(* -----------------------------------------------------------------------------
| This sample has been supplied by Beckhoff As-Is and is intended only as an   |
| example implementation. Functionality is not guaranteed.                     |
----------------------------------------------------------------------------- *)

FUNCTION_BLOCK FB_CorkingRotation
VAR_INPUT
	bExecute : BOOL;
	bLimitSwitch : BOOL;
END_VAR
VAR_OUTPUT
	bRotation : BOOL; 
	bDone : BOOL;
	bError : BOOL;
	nErrId : UDINT;
END_VAR
VAR
	nCnt : UDINT;
END_VAR

(* -----------------------------------------------------------------------------
| This sample has been supplied by Beckhoff As-Is and is intended only as an   |
| example implementation. Functionality is not guaranteed.                     |
----------------------------------------------------------------------------- *)

IF bExecute THEN
	nCnt := nCnt + 1;
	bRotation := (nCnt >= 1 AND nCnt < 100) OR
				(nCnt >= 201 AND nCnt < 300) OR
				(nCnt >= 401 AND nCnt < 500) OR
				(nCnt >= 601 AND nCnt < 700) OR
				(nCnt >= 800 AND nCnt < 1000);
	IF nCnt >= 1000 THEN
		IF bLimitSwitch THEN
			bDone := TRUE;
			bError := FALSE;
			nErrId := 0;
		ELSE
			bDone := FALSE;
			bError := 1;
			nErrId := 16#9999_0001;
		END_IF			
	END_IF
ELSE
	bError := FALSE;
	bRotation := FALSE;
	nCnt := 0;
	bDone := FALSE;
END_IF

END_FUNCTION_BLOCK

(* stored: Version 1.1.0.1, ProductVersion 3.1.4024.12
   POU FB_CorkingRotation: Id {8583df25-4107-4e91-a9c0-f76aea7f674c}, SpecialFunc None *)
